// This function has been automatically generated from the project information.
{attribute 'signature_flag' := '1073741824'}
{attribute 'TcGenerated'}
{attribute 'no-analysis'}
FUNCTION F_GetTitle : WSTRING
VAR_INPUT
	
END_VAR

F_GetTitle := "ExercicesForPlcProgramming";

END_FUNCTION

(* stored: Version 1.1.0.1
   POU F_GetTitle: Id {1051a50d-db37-4d8a-8dcf-e5deb7994024}, SpecialFunc None *)
